(* Logix 5000 project; controller cal1632 1756-L62 rev 16.20; software revision 16.05; part 52 of 57 *)
(* tags used below, declared in another part *)
   FAULT : BOOL;
   HMI : BOOL;
   p01_recipe_active : recipe;
   p01r09_pb_global_reset : BOOL;
   p01r13_line_running : BOOL;
   p01r13_line_slow_ramp : BOOL;
   p02_real_from_hmi : hmi_real;
   p21r10_index_kd : REAL;
   p21r10_index_ki : REAL;
   p21r10_index_kp : REAL;
   p21r11_index_kd : REAL;
   p21r11_index_ki : REAL;
   p21r11_index_kp : REAL;
   p21r11_run_kd : REAL;
   p21r11_run_ki : REAL;
   p21r11_run_kp : REAL;
   p25_ao_selected_speed : REAL;
   p289_di_ss_jog : BOOL;
   p289_di_ss_run : BOOL;
   p29_ai_wa_speed : REAL;
   p29_ai_wa_torque : REAL;
   p29_ai_wb_speed : REAL;
   p29_ai_wb_torque : REAL;
   p29_ai_wdr_lc : REAL;
   p29_di_wdr_a : BOOL;
   p29_di_wdr_index_fwd : BOOL;
   p29_dint_to_hmi : DINT[16];
   p29r08 : routine;
   p29r08_timer_fault : TIMER[4];
   p29r08_timer_warning : TIMER[4];
   p29r09 : routine;
   p29r09_tension_mode : BOOL;
   p29r09_timer_fault : TIMER[4];
   p29r09_timer_warning : TIMER[4];
   p29r09_torque_mode : BOOL;
   p29r09_winder_a_active : BOOL;
   p29r09_winder_b_active : BOOL;
   p29r09_winder_jog : BOOL;
   p29r09_winder_off : BOOL;
   p29r09_winder_run : BOOL;
   p29r10 : routine;
   p29r10_accel_bias : REAL;
   p29r10_calc_speed_offset : REAL;
   p29r10_index_active : BOOL;
   p29r10_misc_index_factor : REAL;
   p29r10_param_psn_gain : REAL;
   p29r10_pid_out : REAL;
   p29r10_pid_psn : PID;
   p29r10_pid_psn_cv : REAL;
   p29r10_pid_psn_pv : REAL;
   p29r10_pid_torque : REAL;
   p29r10_pid_tq : PID;
   p29r10_pid_tq_cv : REAL;
   p29r10_psn_gain : REAL;
   p29r10_request_run : BOOL;
   p29r10_run_permissive : BOOL;
   p29r10_speed_offset : REAL;
   p29r10_timer : TIMER[4];
   p29r10_timer_fault : TIMER[4];
   p29r10_timer_warning : TIMER[4];
   p29r11 : routine;
   p29r11_accel_bias : REAL;
   p29r11_calc_speed_offset : REAL;
   p29r11_index_active : BOOL;
   p29r11_misc_index_factor : REAL;
   p29r11_param_psn_gain : REAL;
   p29r11_pid_out : REAL;
   p29r11_pid_psn : PID;
   p29r11_pid_psn_cv : REAL;
   p29r11_pid_psn_pv : REAL;
   p29r11_pid_torque : REAL;
   p29r11_pid_tq : PID;
   p29r11_pid_tq_cv : REAL;
   p29r11_psn_gain : REAL;
   p29r11_request_run : BOOL;
   p29r11_run_permissive : BOOL;
   p29r11_speed_offset : REAL;
   p29r11_timer : TIMER[1];
   p29r11_timer_fault : TIMER[4];
   p29r11_timer_warning : TIMER[4];
   p29r15 : routine;
   p29r15_state : DINT;
   p29r15_wdra_active : BOOL;
   p29r16 : routine;
   p29r16_state : DINT;
   p29r16_wdrb_active : BOOL;
   p29r20 : routine;
(* P29_Winder, continued *)

ROUTINE R08_Warnings   (* ladder *)
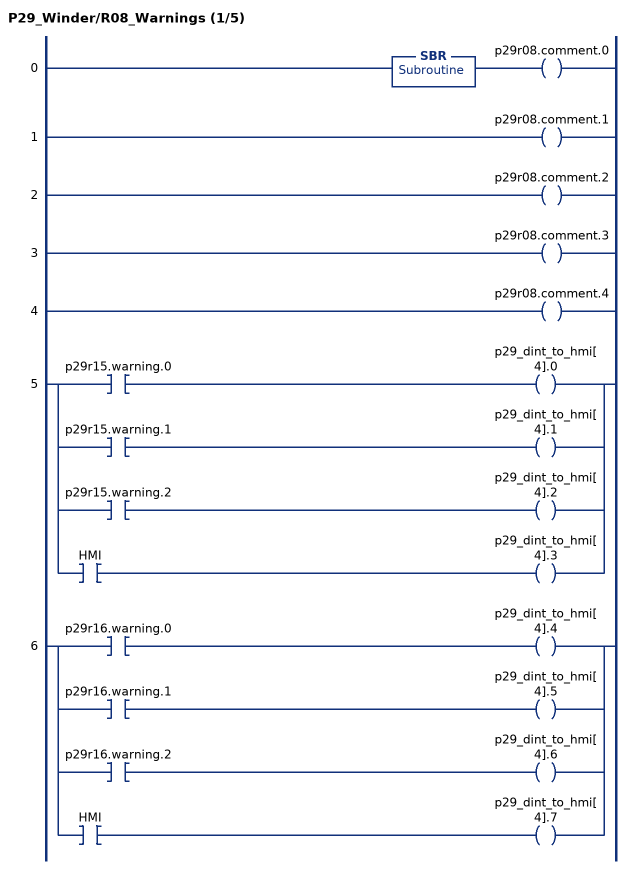
   0: SBR()OTE(p29r08.comment.0);
   1: OTE(p29r08.comment.1);
   2: OTE(p29r08.comment.2);
   3: OTE(p29r08.comment.3);
   4: OTE(p29r08.comment.4);
   5: [XIC(p29r15.warning.0) OTE(p29_dint_to_hmi[4].0) ,XIC(p29r15.warning.1) OTE(p29_dint_to_hmi[4].1) ,XIC(p29r15.warning.2) OTE(p29_dint_to_hmi[4].2) ,XIC(HMI) OTE(p29_dint_to_hmi[4].3) ];
   6: [XIC(p29r16.warning.0) OTE(p29_dint_to_hmi[4].4) ,XIC(p29r16.warning.1) OTE(p29_dint_to_hmi[4].5) ,XIC(p29r16.warning.2) OTE(p29_dint_to_hmi[4].6) ,XIC(HMI) OTE(p29_dint_to_hmi[4].7) ];
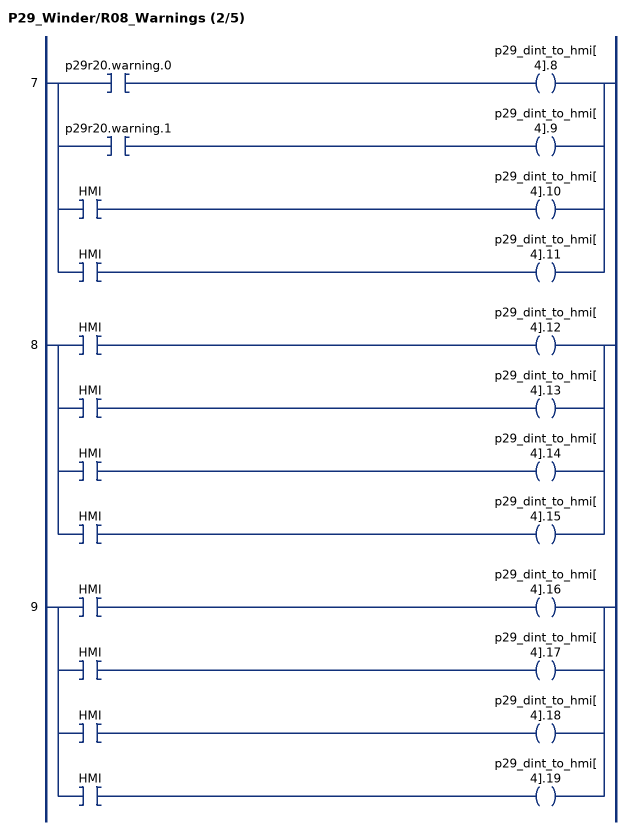
   7: [XIC(p29r20.warning.0) OTE(p29_dint_to_hmi[4].8) ,XIC(p29r20.warning.1) OTE(p29_dint_to_hmi[4].9) ,XIC(HMI) OTE(p29_dint_to_hmi[4].10) ,XIC(HMI) OTE(p29_dint_to_hmi[4].11) ];
   8: [XIC(HMI) OTE(p29_dint_to_hmi[4].12) ,XIC(HMI) OTE(p29_dint_to_hmi[4].13) ,XIC(HMI) OTE(p29_dint_to_hmi[4].14) ,XIC(HMI) OTE(p29_dint_to_hmi[4].15) ];
   9: [XIC(HMI) OTE(p29_dint_to_hmi[4].16) ,XIC(HMI) OTE(p29_dint_to_hmi[4].17) ,XIC(HMI) OTE(p29_dint_to_hmi[4].18) ,XIC(HMI) OTE(p29_dint_to_hmi[4].19) ];
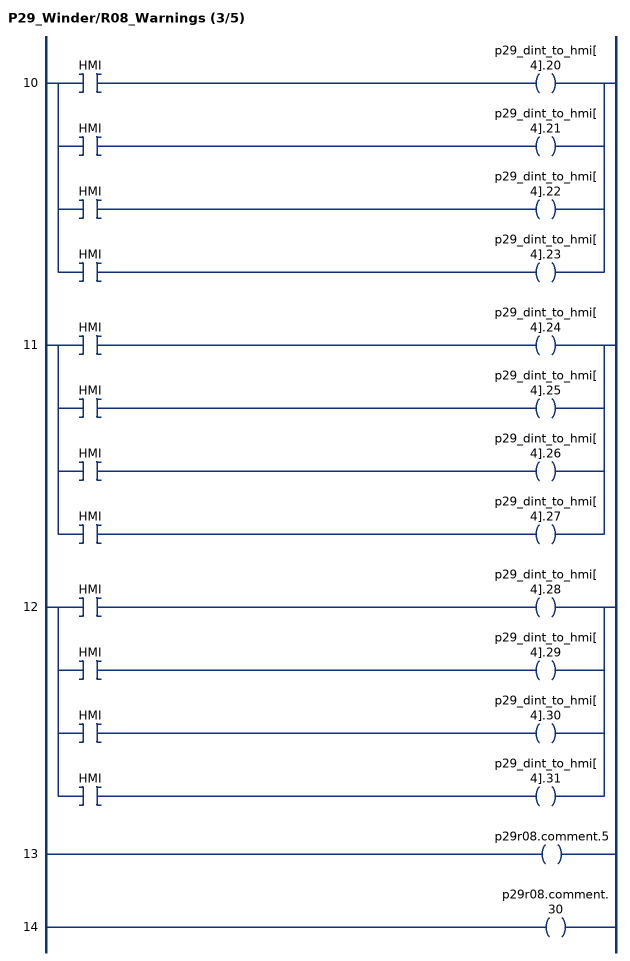
   10: [XIC(HMI) OTE(p29_dint_to_hmi[4].20) ,XIC(HMI) OTE(p29_dint_to_hmi[4].21) ,XIC(HMI) OTE(p29_dint_to_hmi[4].22) ,XIC(HMI) OTE(p29_dint_to_hmi[4].23) ];
   11: [XIC(HMI) OTE(p29_dint_to_hmi[4].24) ,XIC(HMI) OTE(p29_dint_to_hmi[4].25) ,XIC(HMI) OTE(p29_dint_to_hmi[4].26) ,XIC(HMI) OTE(p29_dint_to_hmi[4].27) ];
   12: [XIC(HMI) OTE(p29_dint_to_hmi[4].28) ,XIC(HMI) OTE(p29_dint_to_hmi[4].29) ,XIC(HMI) OTE(p29_dint_to_hmi[4].30) ,XIC(HMI) OTE(p29_dint_to_hmi[4].31) ];
   13: OTE(p29r08.comment.5);
   14: OTE(p29r08.comment.30);
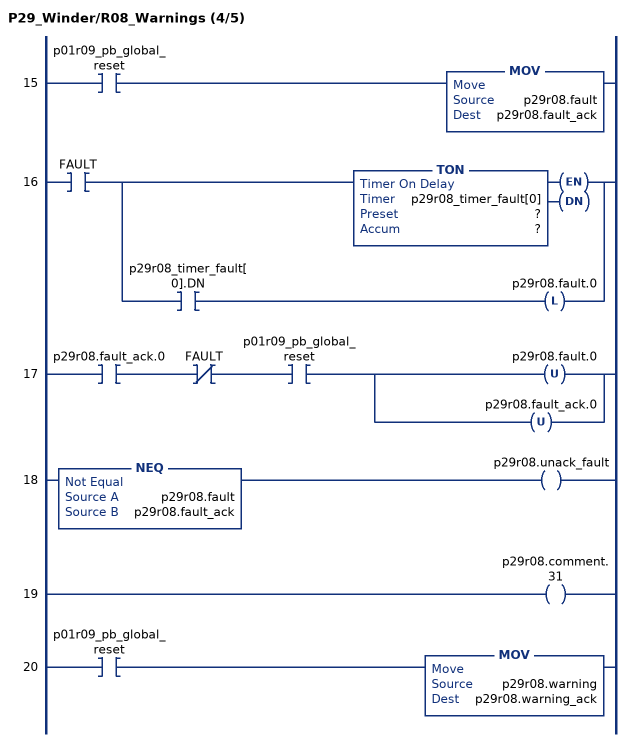
   15: XIC(p01r09_pb_global_reset)MOV(p29r08.fault,p29r08.fault_ack);
   16: XIC(FAULT)[TON(p29r08_timer_fault[0],?,?) ,XIC(p29r08_timer_fault[0].DN) OTL(p29r08.fault.0) ];
   17: XIC(p29r08.fault_ack.0)XIO(FAULT)XIC(p01r09_pb_global_reset)[OTU(p29r08.fault.0) ,OTU(p29r08.fault_ack.0) ];
   18: NEQ(p29r08.fault,p29r08.fault_ack)OTE(p29r08.unack_fault);
   19: OTE(p29r08.comment.31);
   20: XIC(p01r09_pb_global_reset)MOV(p29r08.warning,p29r08.warning_ack);
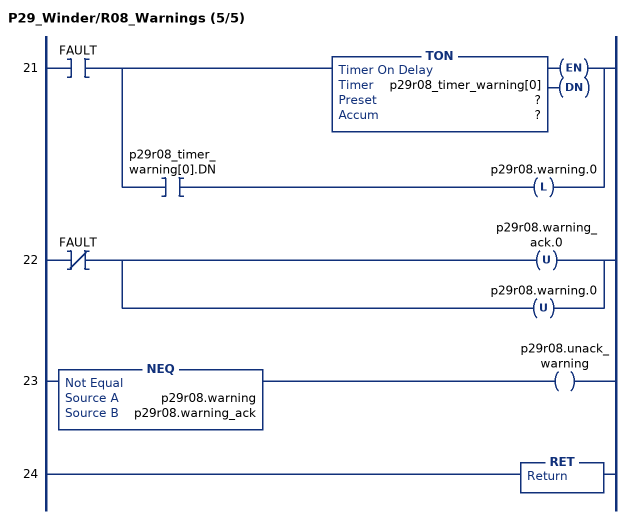
   21: XIC(FAULT)[TON(p29r08_timer_warning[0],?,?) ,XIC(p29r08_timer_warning[0].DN) OTL(p29r08.warning.0) ];
   22: XIO(FAULT)[OTU(p29r08.warning_ack.0) ,OTU(p29r08.warning.0) ];
   23: NEQ(p29r08.warning,p29r08.warning_ack)OTE(p29r08.unack_warning);
   24: RET();
END_ROUTINE

ROUTINE R09_Modes   (* ladder *)
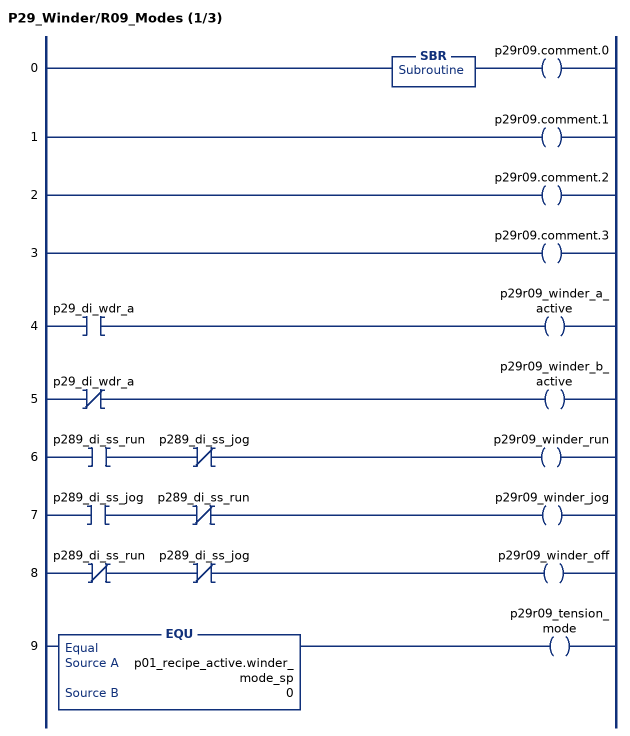
   0: SBR()OTE(p29r09.comment.0);
   1: OTE(p29r09.comment.1);
   2: OTE(p29r09.comment.2);
   3: OTE(p29r09.comment.3);
   4: XIC(p29_di_wdr_a)OTE(p29r09_winder_a_active);
   5: XIO(p29_di_wdr_a)OTE(p29r09_winder_b_active);
   6: XIC(p289_di_ss_run)XIO(p289_di_ss_jog)OTE(p29r09_winder_run);
   7: XIC(p289_di_ss_jog)XIO(p289_di_ss_run)OTE(p29r09_winder_jog);
   8: XIO(p289_di_ss_run)XIO(p289_di_ss_jog)OTE(p29r09_winder_off);
   9: EQU(p01_recipe_active.winder_mode_sp,0)OTE(p29r09_tension_mode);
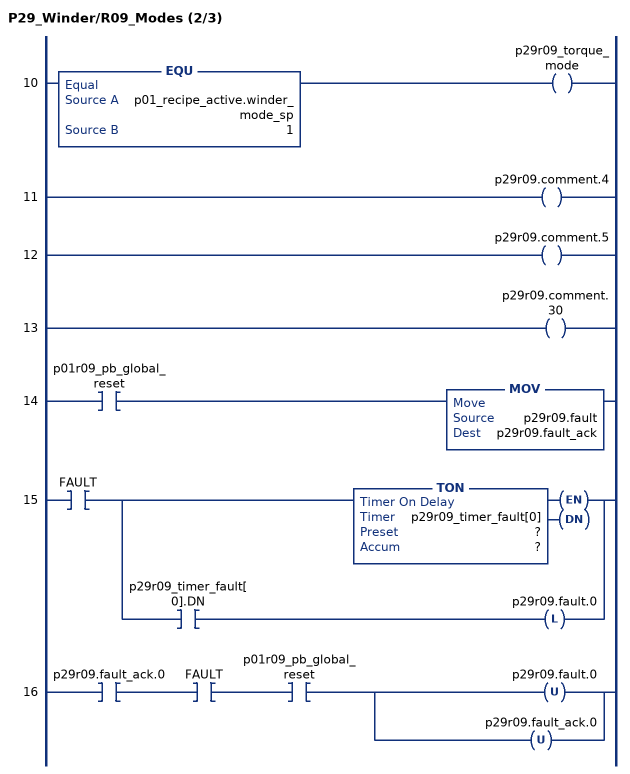
   10: EQU(p01_recipe_active.winder_mode_sp,1)OTE(p29r09_torque_mode);
   11: OTE(p29r09.comment.4);
   12: OTE(p29r09.comment.5);
   13: OTE(p29r09.comment.30);
   14: XIC(p01r09_pb_global_reset)MOV(p29r09.fault,p29r09.fault_ack);
   15: XIC(FAULT)[TON(p29r09_timer_fault[0],?,?) ,XIC(p29r09_timer_fault[0].DN) OTL(p29r09.fault.0) ];
   16: XIC(p29r09.fault_ack.0)XIC(FAULT)XIC(p01r09_pb_global_reset)[OTU(p29r09.fault.0) ,OTU(p29r09.fault_ack.0) ];
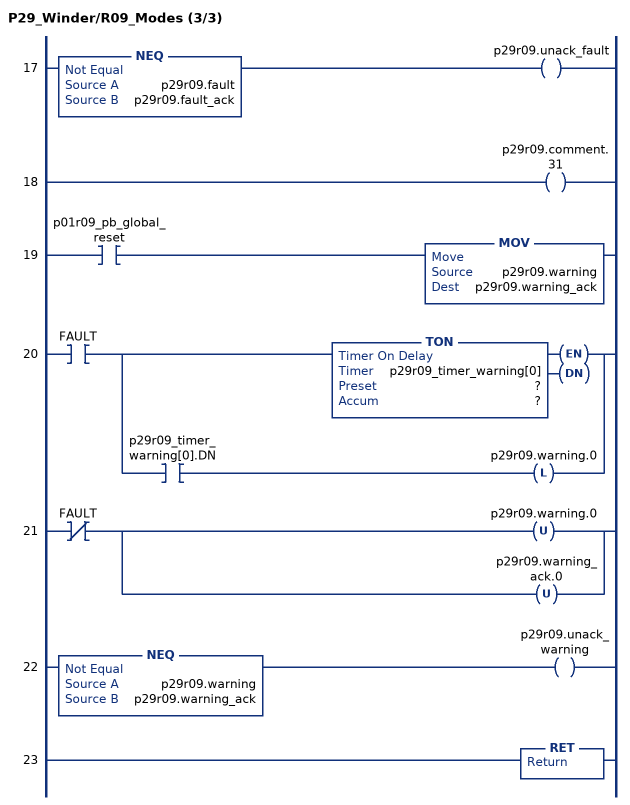
   17: NEQ(p29r09.fault,p29r09.fault_ack)OTE(p29r09.unack_fault);
   18: OTE(p29r09.comment.31);
   19: XIC(p01r09_pb_global_reset)MOV(p29r09.warning,p29r09.warning_ack);
   20: XIC(FAULT)[TON(p29r09_timer_warning[0],?,?) ,XIC(p29r09_timer_warning[0].DN) OTL(p29r09.warning.0) ];
   21: XIO(FAULT)[OTU(p29r09.warning.0) ,OTU(p29r09.warning_ack.0) ];
   22: NEQ(p29r09.warning,p29r09.warning_ack)OTE(p29r09.unack_warning);
   23: RET();
END_ROUTINE

ROUTINE R10_Winder_A_Speed_Control   (* ladder *)
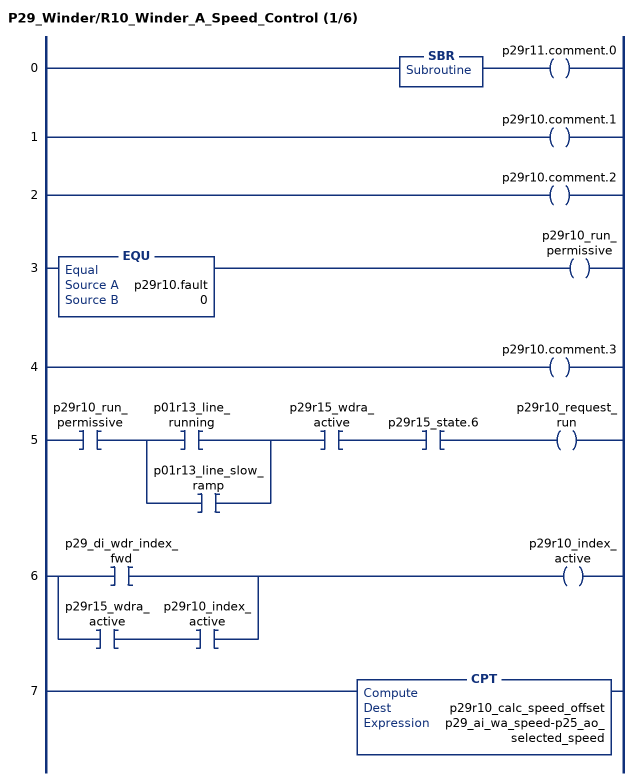
   0: SBR()OTE(p29r11.comment.0);
   1: OTE(p29r10.comment.1);
   2: OTE(p29r10.comment.2);
   3: EQU(p29r10.fault,0)OTE(p29r10_run_permissive);
   4: OTE(p29r10.comment.3);
   5: XIC(p29r10_run_permissive)[XIC(p01r13_line_running) ,XIC(p01r13_line_slow_ramp) ]XIC(p29r15_wdra_active)XIC(p29r15_state.6)OTE(p29r10_request_run);
   6: [XIC(p29_di_wdr_index_fwd) ,XIC(p29r15_wdra_active) XIC(p29r10_index_active) ]OTE(p29r10_index_active);
   7: CPT(p29r10_calc_speed_offset,p29_ai_wa_speed-p25_ao_selected_speed);
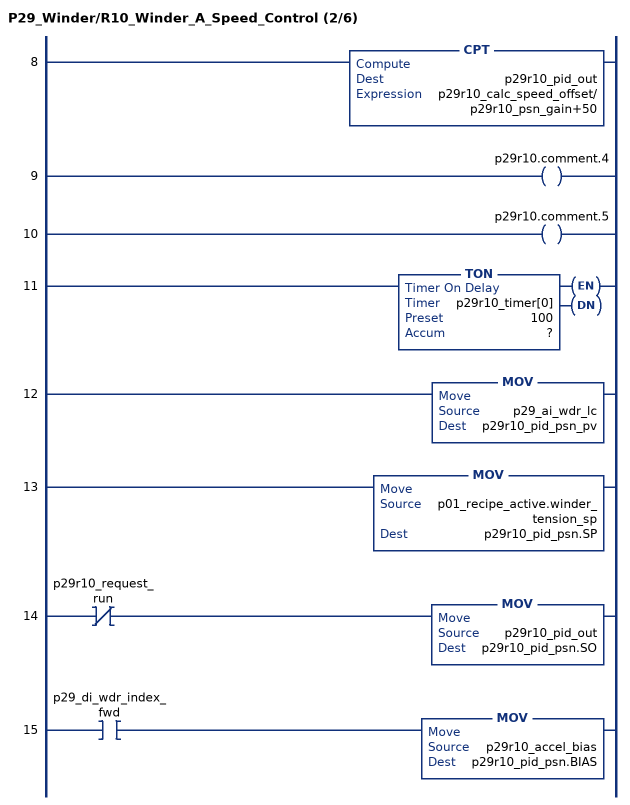
   8: CPT(p29r10_pid_out,p29r10_calc_speed_offset/p29r10_psn_gain+50);
   9: OTE(p29r10.comment.4);
   10: OTE(p29r10.comment.5);
   11: TON(p29r10_timer[0],?,?);
   12: MOV(p29_ai_wdr_lc,p29r10_pid_psn_pv);
   13: MOV(p01_recipe_active.winder_tension_sp,p29r10_pid_psn.SP);
   14: XIO(p29r10_request_run)MOV(p29r10_pid_out,p29r10_pid_psn.SO);
   15: XIC(p29_di_wdr_index_fwd)MOV(p29r10_accel_bias,p29r10_pid_psn.BIAS);
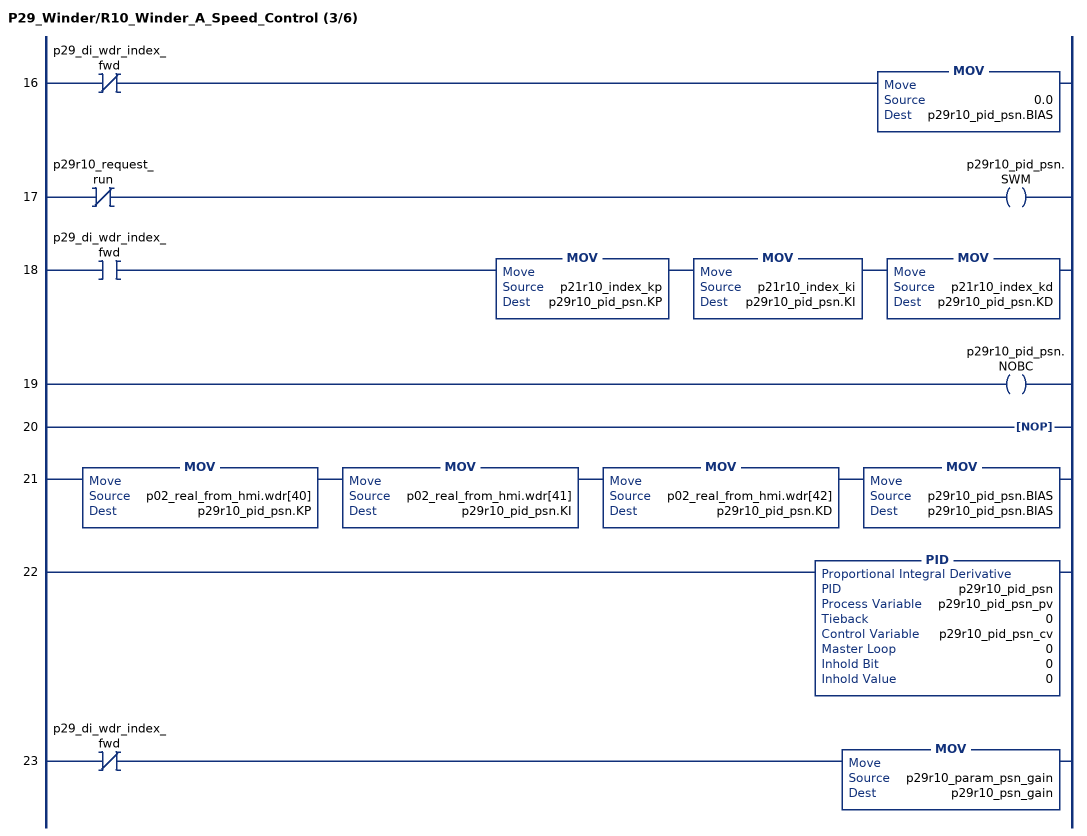
   16: XIO(p29_di_wdr_index_fwd)MOV(0.0,p29r10_pid_psn.BIAS);
   17: XIO(p29r10_request_run)OTE(p29r10_pid_psn.SWM);
   18: XIC(p29_di_wdr_index_fwd)MOV(p21r10_index_kp,p29r10_pid_psn.KP)MOV(p21r10_index_ki,p29r10_pid_psn.KI)MOV(p21r10_index_kd,p29r10_pid_psn.KD);
   19: OTE(p29r10_pid_psn.NOBC);
   20: NOP();
   21: MOV(p02_real_from_hmi.wdr[40],p29r10_pid_psn.KP)MOV(p02_real_from_hmi.wdr[41],p29r10_pid_psn.KI)MOV(p02_real_from_hmi.wdr[42],p29r10_pid_psn.KD)MOV(p29r10_pid_psn.BIAS,p29r10_pid_psn.BIAS);
   22: PID(p29r10_pid_psn,p29r10_pid_psn_pv,0,p29r10_pid_psn_cv,0,0,0);
   23: XIO(p29_di_wdr_index_fwd)MOV(p29r10_param_psn_gain,p29r10_psn_gain);
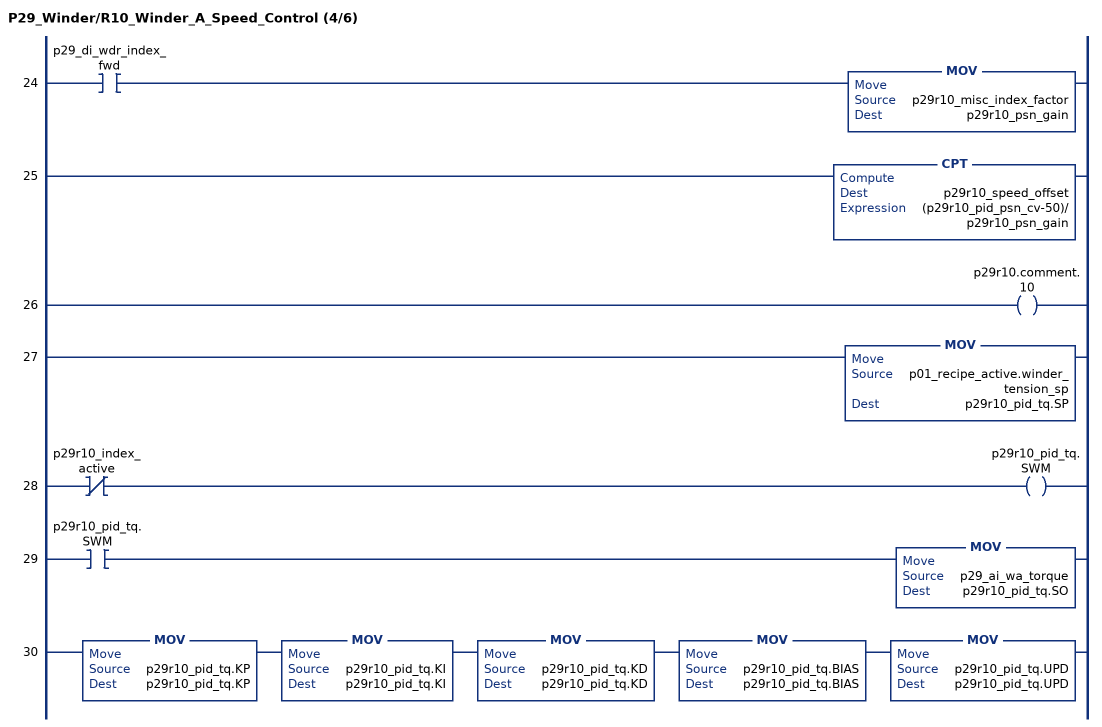
   24: XIC(p29_di_wdr_index_fwd)MOV(p29r10_misc_index_factor,p29r10_psn_gain);
   25: CPT(p29r10_speed_offset,(p29r10_pid_psn_cv-50)/p29r10_psn_gain);
   26: OTE(p29r10.comment.10);
   27: MOV(p01_recipe_active.winder_tension_sp,p29r10_pid_tq.SP);
   28: XIO(p29r10_index_active)OTE(p29r10_pid_tq.SWM);
   29: XIC(p29r10_pid_tq.SWM)MOV(p29_ai_wa_torque,p29r10_pid_tq.SO);
   30: MOV(p29r10_pid_tq.KP,p29r10_pid_tq.KP)MOV(p29r10_pid_tq.KI,p29r10_pid_tq.KI)MOV(p29r10_pid_tq.KD,p29r10_pid_tq.KD)MOV(p29r10_pid_tq.BIAS,p29r10_pid_tq.BIAS)MOV(p29r10_pid_tq.UPD,p29r10_pid_tq.UPD);
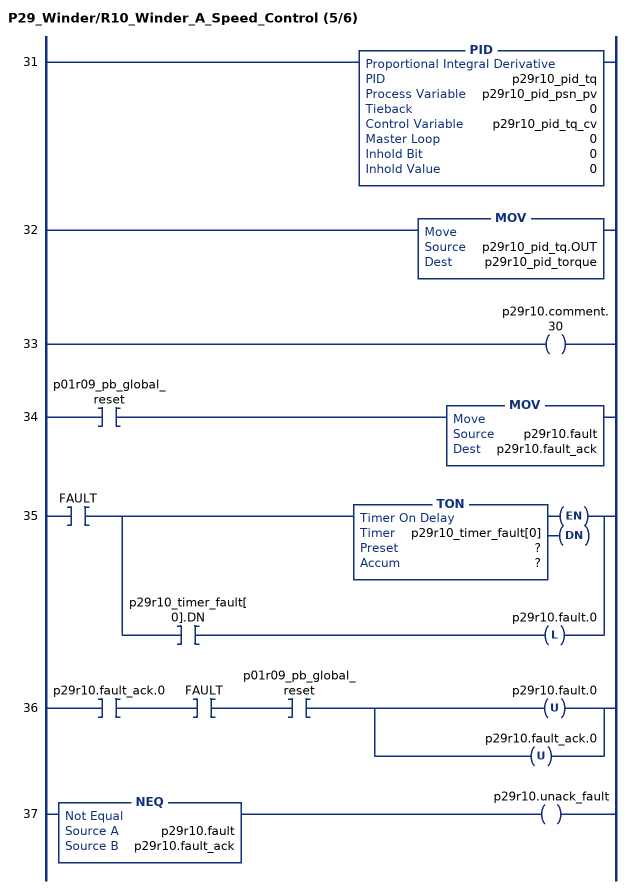
   31: PID(p29r10_pid_tq,p29r10_pid_psn_pv,0,p29r10_pid_tq_cv,0,0,0);
   32: MOV(p29r10_pid_tq.OUT,p29r10_pid_torque);
   33: OTE(p29r10.comment.30);
   34: XIC(p01r09_pb_global_reset)MOV(p29r10.fault,p29r10.fault_ack);
   35: XIC(FAULT)[TON(p29r10_timer_fault[0],?,?) ,XIC(p29r10_timer_fault[0].DN) OTL(p29r10.fault.0) ];
   36: XIC(p29r10.fault_ack.0)XIC(FAULT)XIC(p01r09_pb_global_reset)[OTU(p29r10.fault.0) ,OTU(p29r10.fault_ack.0) ];
   37: NEQ(p29r10.fault,p29r10.fault_ack)OTE(p29r10.unack_fault);
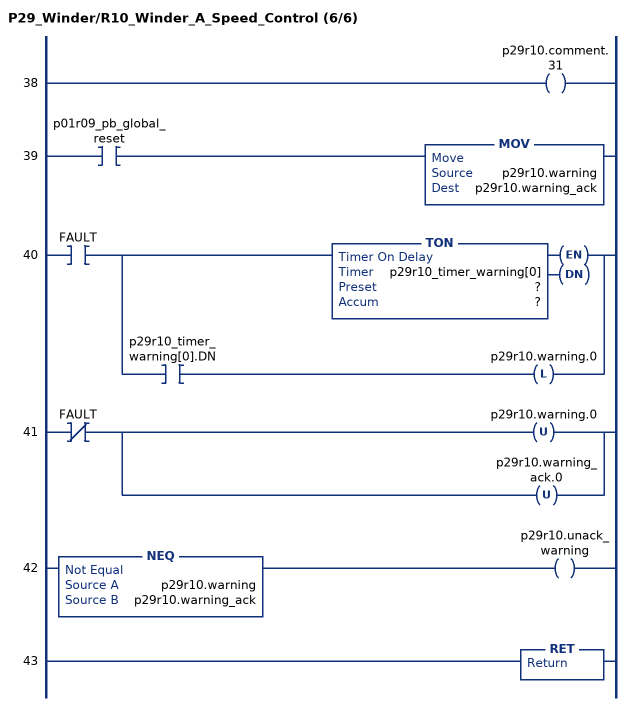
   38: OTE(p29r10.comment.31);
   39: XIC(p01r09_pb_global_reset)MOV(p29r10.warning,p29r10.warning_ack);
   40: XIC(FAULT)[TON(p29r10_timer_warning[0],?,?) ,XIC(p29r10_timer_warning[0].DN) OTL(p29r10.warning.0) ];
   41: XIO(FAULT)[OTU(p29r10.warning.0) ,OTU(p29r10.warning_ack.0) ];
   42: NEQ(p29r10.warning,p29r10.warning_ack)OTE(p29r10.unack_warning);
   43: RET();
END_ROUTINE

ROUTINE R11_Winder_B_Speed_Control   (* ladder *)
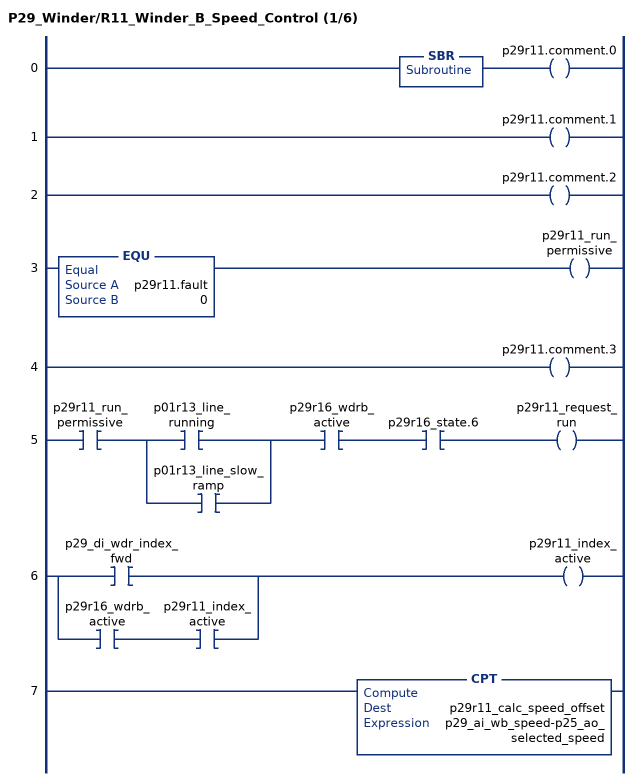
   0: SBR()OTE(p29r11.comment.0);
   1: OTE(p29r11.comment.1);
   2: OTE(p29r11.comment.2);
   3: EQU(p29r11.fault,0)OTE(p29r11_run_permissive);
   4: OTE(p29r11.comment.3);
   5: XIC(p29r11_run_permissive)[XIC(p01r13_line_running) ,XIC(p01r13_line_slow_ramp) ]XIC(p29r16_wdrb_active)XIC(p29r16_state.6)OTE(p29r11_request_run);
   6: [XIC(p29_di_wdr_index_fwd) ,XIC(p29r16_wdrb_active) XIC(p29r11_index_active) ]OTE(p29r11_index_active);
   7: CPT(p29r11_calc_speed_offset,p29_ai_wb_speed-p25_ao_selected_speed);
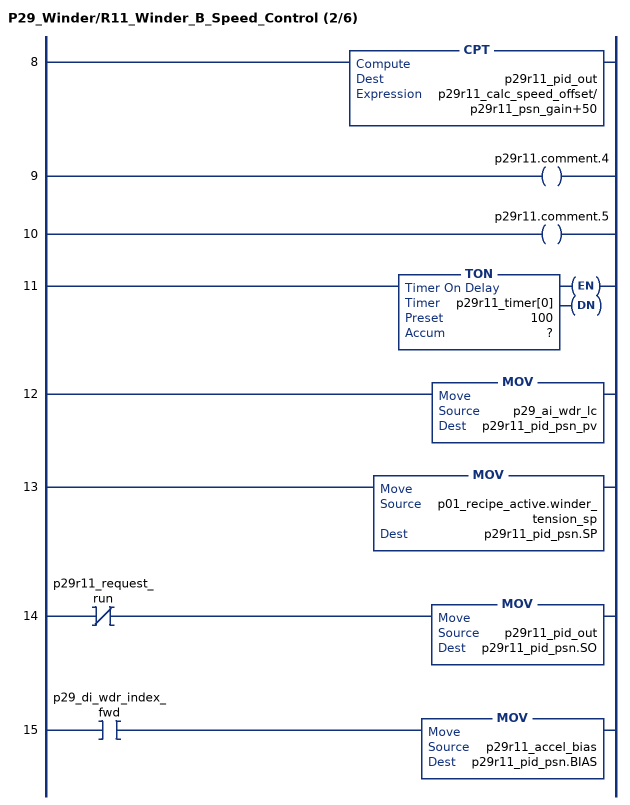
   8: CPT(p29r11_pid_out,p29r11_calc_speed_offset/p29r11_psn_gain+50);
   9: OTE(p29r11.comment.4);
   10: OTE(p29r11.comment.5);
   11: TON(p29r11_timer[0],?,?);
   12: MOV(p29_ai_wdr_lc,p29r11_pid_psn_pv);
   13: MOV(p01_recipe_active.winder_tension_sp,p29r11_pid_psn.SP);
   14: XIO(p29r11_request_run)MOV(p29r11_pid_out,p29r11_pid_psn.SO);
   15: XIC(p29_di_wdr_index_fwd)MOV(p29r11_accel_bias,p29r11_pid_psn.BIAS);
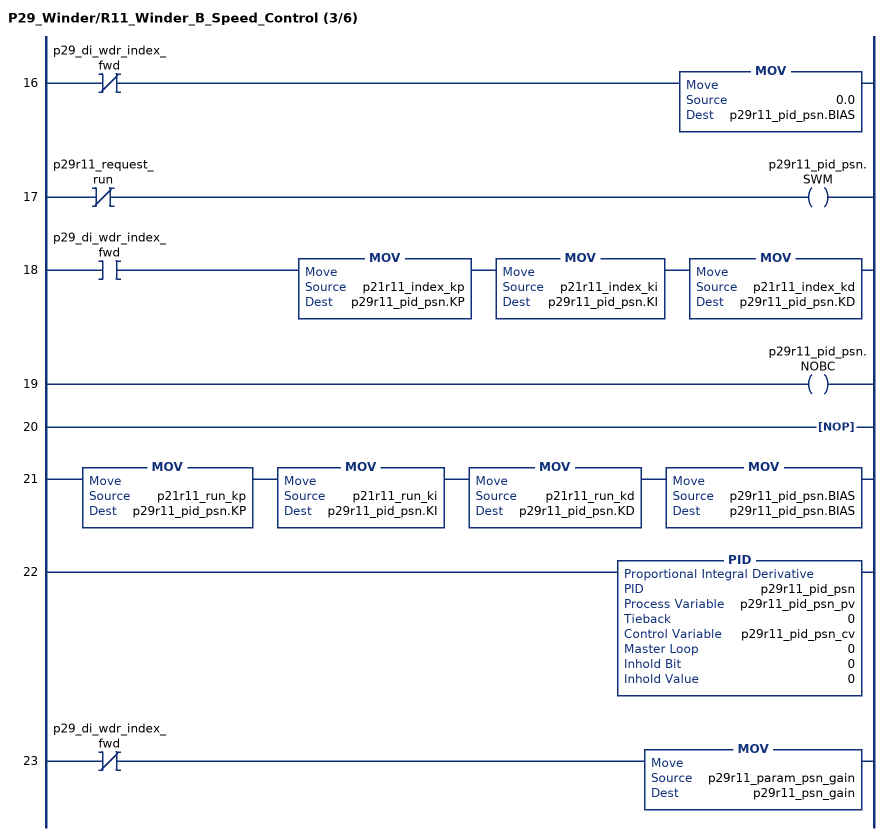
   16: XIO(p29_di_wdr_index_fwd)MOV(0.0,p29r11_pid_psn.BIAS);
   17: XIO(p29r11_request_run)OTE(p29r11_pid_psn.SWM);
   18: XIC(p29_di_wdr_index_fwd)MOV(p21r11_index_kp,p29r11_pid_psn.KP)MOV(p21r11_index_ki,p29r11_pid_psn.KI)MOV(p21r11_index_kd,p29r11_pid_psn.KD);
   19: OTE(p29r11_pid_psn.NOBC);
   20: NOP();
   21: MOV(p21r11_run_kp,p29r11_pid_psn.KP)MOV(p21r11_run_ki,p29r11_pid_psn.KI)MOV(p21r11_run_kd,p29r11_pid_psn.KD)MOV(p29r11_pid_psn.BIAS,p29r11_pid_psn.BIAS);
   22: PID(p29r11_pid_psn,p29r11_pid_psn_pv,0,p29r11_pid_psn_cv,0,0,0);
   23: XIO(p29_di_wdr_index_fwd)MOV(p29r11_param_psn_gain,p29r11_psn_gain);
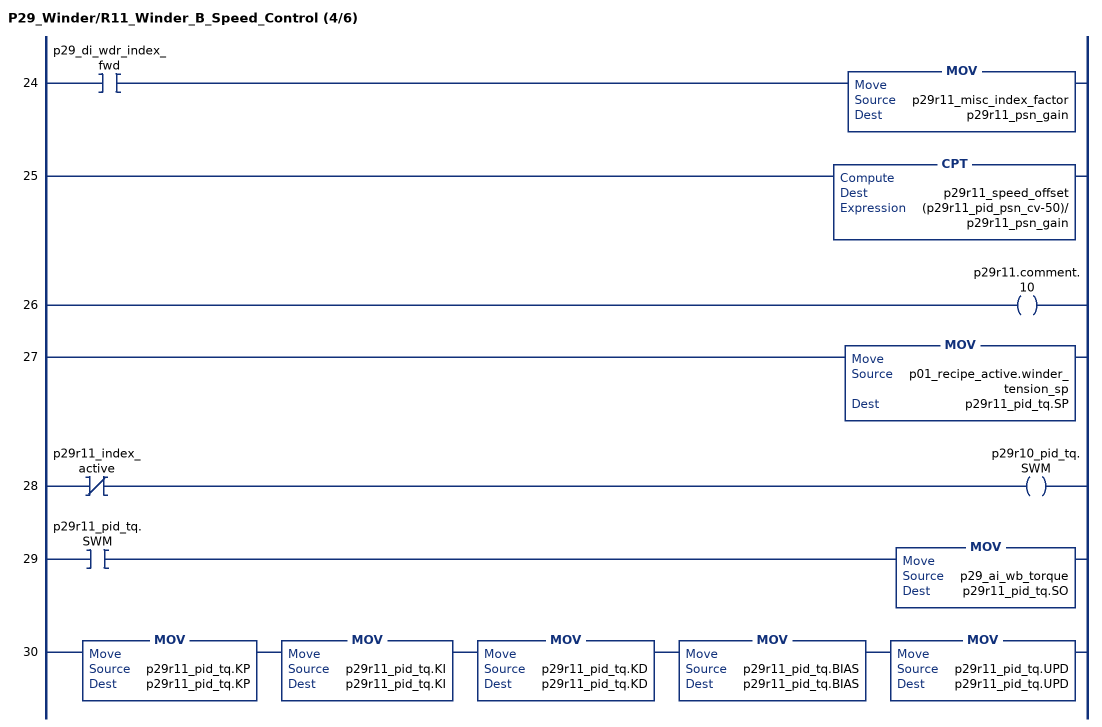
   24: XIC(p29_di_wdr_index_fwd)MOV(p29r11_misc_index_factor,p29r11_psn_gain);
   25: CPT(p29r11_speed_offset,(p29r11_pid_psn_cv-50)/p29r11_psn_gain);
   26: OTE(p29r11.comment.10);
   27: MOV(p01_recipe_active.winder_tension_sp,p29r11_pid_tq.SP);
   28: XIO(p29r11_index_active)OTE(p29r10_pid_tq.SWM);
   29: XIC(p29r11_pid_tq.SWM)MOV(p29_ai_wb_torque,p29r11_pid_tq.SO);
   30: MOV(p29r11_pid_tq.KP,p29r11_pid_tq.KP)MOV(p29r11_pid_tq.KI,p29r11_pid_tq.KI)MOV(p29r11_pid_tq.KD,p29r11_pid_tq.KD)MOV(p29r11_pid_tq.BIAS,p29r11_pid_tq.BIAS)MOV(p29r11_pid_tq.UPD,p29r11_pid_tq.UPD);
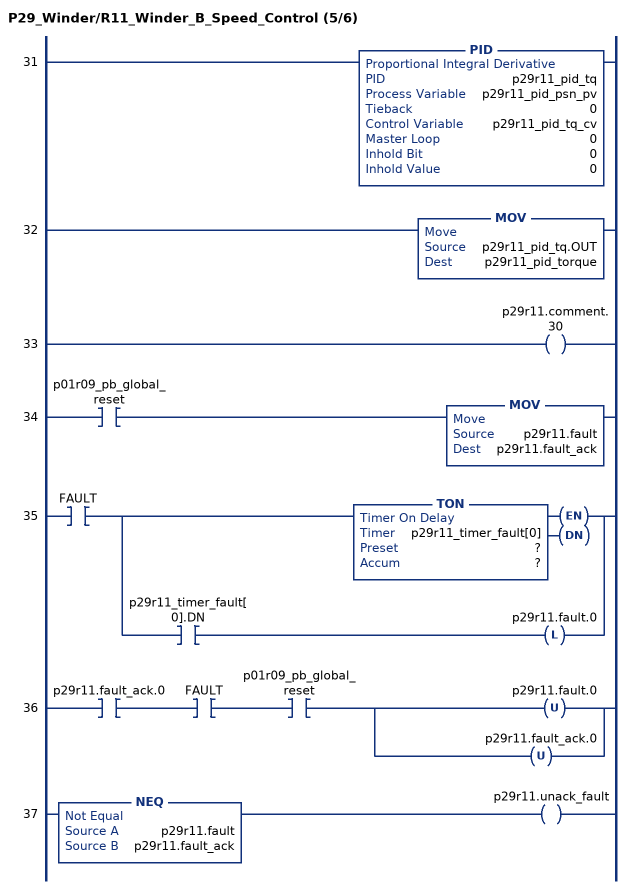
   31: PID(p29r11_pid_tq,p29r11_pid_psn_pv,0,p29r11_pid_tq_cv,0,0,0);
   32: MOV(p29r11_pid_tq.OUT,p29r11_pid_torque);
   33: OTE(p29r11.comment.30);
   34: XIC(p01r09_pb_global_reset)MOV(p29r11.fault,p29r11.fault_ack);
   35: XIC(FAULT)[TON(p29r11_timer_fault[0],?,?) ,XIC(p29r11_timer_fault[0].DN) OTL(p29r11.fault.0) ];
   36: XIC(p29r11.fault_ack.0)XIC(FAULT)XIC(p01r09_pb_global_reset)[OTU(p29r11.fault.0) ,OTU(p29r11.fault_ack.0) ];
   37: NEQ(p29r11.fault,p29r11.fault_ack)OTE(p29r11.unack_fault);
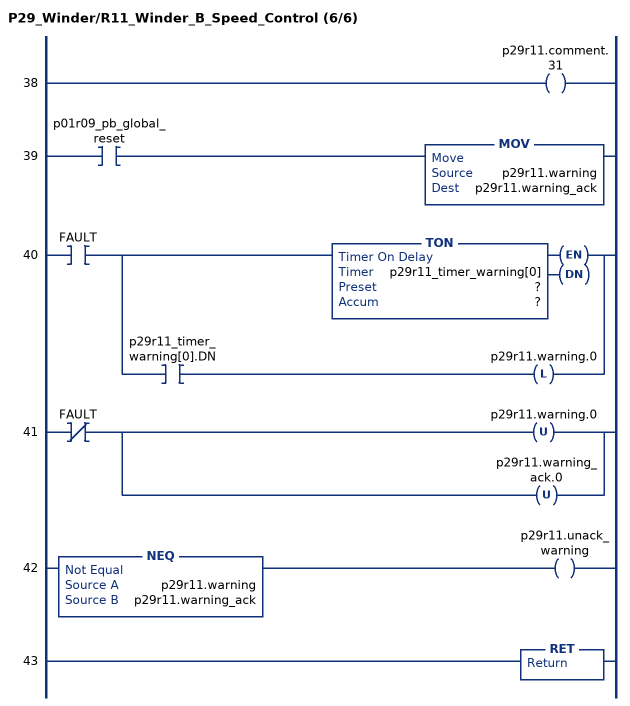
   38: OTE(p29r11.comment.31);
   39: XIC(p01r09_pb_global_reset)MOV(p29r11.warning,p29r11.warning_ack);
   40: XIC(FAULT)[TON(p29r11_timer_warning[0],?,?) ,XIC(p29r11_timer_warning[0].DN) OTL(p29r11.warning.0) ];
   41: XIO(FAULT)[OTU(p29r11.warning.0) ,OTU(p29r11.warning_ack.0) ];
   42: NEQ(p29r11.warning,p29r11.warning_ack)OTE(p29r11.unack_warning);
   43: RET();
END_ROUTINE
